FUNCTION_BLOCK FB_OpenLoopControl
VAR_INPUT

	bEnable : BOOL;
	fVelocityRef : REAL;
	fQMax : LREAL;

END_VAR
VAR_OUTPUT
	fValveOutput_openLoopControl : LREAL;
END_VAR
VAR
	Bore_Area : LREAL := 0.0033183;
	Annulus_Area : LREAL := 0.002356;
	
END_VAR



IF bEnable = TRUE THEN
	
	IF fVelocityRef > 0 THEN
		
		fValveOutput_openLoopControl := (fVelocityRef * Bore_Area * 60000) / fQMax;
	
	ELSE
		fValveOutput_openLoopControl := (fVelocityRef * Annulus_Area  * 60000) / fQMax;
		
	END_IF

ELSE
	
	fValveOutput_openLoopControl := 0;
	
	
END_IF

END_FUNCTION_BLOCK

(* stored: Version 1.1.0.1, ProductVersion 3.1.4024.10
   POU FB_OpenLoopControl: Id {bbc24abb-6cdb-48e4-8aee-fd9b7593f3dd}, SpecialFunc None *)
